FUNCTION_BLOCK FB_ParamMediatorDmax IMPLEMENTS I_ParamMediator
VAR
  _pCreateWorker : POINTER TO FB_WorkerDefGrid_Python;
  _pCamWorker : POINTER TO FB_WorkerDefGrid_Camera;
  _pDefWorker : POINTER TO FB_WorkerDefGrid_Deformation;
  bInitOk     : BOOL;
END_VAR

(*
  Release deformation ct
  TODO: find another way to do inter worker communication for generic methods.
*)
METHOD ClearCachedCT
VAR_INPUT
  iCT              : I_CT;
END_VAR
IF bInitOk THEN
  _pCreateWorker^.DeleteDefCt(iCT:=iCT);
END_IF
END_METHOD

{attribute 'monitoring':='call'}
PROPERTY fCameraToPrintOffset : LREAL
GET
IF bInitOk THEN
  fCameraToPrintOffset := _pCamWorker^.fCameraToPrintOffset;
END_IF
END_GET
END_PROPERTY

{attribute 'monitoring':='call'}
PROPERTY fDetectToCamera : LREAL
GET
fDetectToCamera := _pCamWorker^.fDetectToCamOffset;
END_GET
END_PROPERTY

(*
  Distance (Offset) from Master-Trigger to Master Reference Position.
  NOTE: This is normally the distance between the first (MASTER) StartPosDetection to first print Module (Printing Unit) 
*)
PROPERTY fMasterDetectToRefPos : LREAL
GET
IF bInitOk THEN
  fMasterDetectToRefPos := _pCamWorker^.fDetectToCamOffset + _pCamWorker^.fCameraToPrintOffset;
END_IF
END_GET
END_PROPERTY

METHOD init
VAR_INPUT
  pCreateWorker : POINTER TO FB_WorkerDefGrid_Python;
  pCamWorker : POINTER TO FB_WorkerDefGrid_Camera;
  pDefWorker : POINTER TO FB_WorkerDefGrid_Deformation;
END_VAR
IF pCamWorker <> 0 AND pCamWorker <>0 AND pCreateWorker <> 0 THEN
  _pCreateWorker := pCreateWorker;
  _pCamWorker := pCamWorker;
  _pDefWorker := pDefWorker;
  bInitOk := TRUE;
END_IF
END_METHOD

PROPERTY sCameraGridSettings : ST_CameraGridSettings
GET
IF bInitOk THEN
  sCameraGridSettings := _pCamWorker^.sCameraGridSettings;
END_IF
END_GET
END_PROPERTY

PROPERTY sDeformationGridSetttings : ST_DefGridSettings
GET
IF bInitOk THEN
  sDeformationGridSetttings := _pDefWorker^.sDeformationGridSettings;
END_IF
END_GET
END_PROPERTY

END_FUNCTION_BLOCK

(* stored: Version 1.1.0.1, ProductVersion 3.1.4024.11
   POU FB_ParamMediatorDmax: Id {9642270e-d441-4770-907b-3f0d0f5dc2e9}, SpecialFunc None
   Folder I_ParamMediator: Id {39f9222d-d28f-4df1-8ed1-e2b3d113f34f}
   Method ClearCachedCT: Id {d54eef11-94fc-4211-8079-b54bc203d3ec}
   Property fCameraToPrintOffset: Id {43edb161-94bb-440e-a146-2ecc3ab0b15d}
   Get Get: Id {687dfcbd-6ad8-4ffb-a3c4-66b35289f9de}
   Property fDetectToCamera: Id {0268497d-c5b0-4639-a734-da6955c88aff}
   Get Get: Id {038181c1-f283-429a-835f-ddc555554d78}
   Property fMasterDetectToRefPos: Id {eee430db-38d9-467a-a866-93af7f37bbbb}
   Get Get: Id {706a4f09-3937-46b5-9660-12df944552bc}
   Method init: Id {9cdfcac0-144a-4d88-8e7f-21c6ce0c82c3}
   Property sCameraGridSettings: Id {686354aa-821c-4c68-8c9d-dafadf8ef6fd}
   Get Get: Id {7a8afb02-f662-4c02-aebf-6b3bd22fae1a}
   Property sDeformationGridSetttings: Id {9cf3f096-207d-452b-ace7-3769f0678220}
   Get Get: Id {f92cba8c-0a7c-4567-a017-f6ac55645e3a} *)
